FUNCTION_BLOCK BaseComponent
VAR_INPUT
END_VAR
VAR_OUTPUT
END_VAR
VAR
	// Time
	ComponentTime: FB_Get_Unix_Timestamp;
	timestamp: ULINT;
END_VAR

METHOD Run : BOOL
VAR_INPUT
END_VAR
END_METHOD

END_FUNCTION_BLOCK

(* stored: Version 1.1.0.1, ProductVersion 3.1.4024.6
   POU BaseComponent: Id {5253bd62-43a4-4dc5-9a8b-6d09f9b444a3}, SpecialFunc None
   Method Run: Id {98d864d5-0f16-4162-8981-2d6b46d665dc} *)
